//Placeholder, WIP --> need to define what purpose this struct serves
TYPE ST_TableNumber :
STRUCT
    In: ST_TableNumberIn;
    Out: ST_TableNumberOut;
END_STRUCT
END_TYPE

(* stored: Version 1.1.0.1
   DUT ST_TableNumber: Id {4dd76721-8462-08bc-2b19-c2901eeab2b7} *)
